// TIA Portal V20 export
DATA_BLOCK "100_CommunicationPLC"   // DB107
// stored: MemoryReserve 100
   VAR
      MotionToPLC : "LER_typeMotionToPLC";
      PLCToMotion : "LER_typePLCToMotion";
   END_VAR
BEGIN
END_DATA_BLOCK
